FUNCTION_BLOCK FB_Parameters_Store IMPLEMENTS If_Parameters
VAR_INPUT PERSISTENT
	Pars	: dt_Parameters;
END_VAR

PROPERTY Par : REFERENCE TO dt_Parameters
GET

Par REF= Pars;
END_GET
END_PROPERTY

END_FUNCTION_BLOCK

(* stored: Version 1.1.0.1, ProductVersion 3.1.4024.15
   POU FB_Parameters_Store: Id {e50436de-36d4-4612-b3d9-7a590fd3e2fa}, SpecialFunc None
   Property Par: Id {b6299f29-3fb6-4083-a3f4-610d1f2debc8}
   Get Get: Id {51efd108-ddcc-489a-89ac-2aeadb0557a7} *)
